// TIA Portal V19 export
DATA_BLOCK "A0301_Ribaltatore_PERS"   // DB58
// stored: MemoryReserve 100
   VAR RETAIN
      Par_Manu : "Positioning_EPOS_Machine_Par";
      Par_Aut : "A0301_Mach_Ribaltatore_Par";
   END_VAR
   VAR
      Par_Aut_Vel : Struct
         Pos1_Frw : LReal := 5000.0;
         Pos2_Frw : LReal := 5000.0;
         Pos0_Brw : LReal := 60000.0;
      END_STRUCT;
   END_VAR
   VAR RETAIN
      Pers_Data : Struct
         EncoderAbsolute_Preset_OK : Bool := TRUE;
         Persistent_ActualPosition : LReal := 2.0;
      END_STRUCT;
   END_VAR
BEGIN
   Par_Manu.PosTolerance := 0.5;
   Par_Manu.DelayInPosition := T#100MS;
   Par_Manu.Man_Vel := 15000.0;
   Par_Manu.Man_Acc := 1000.0;
   Par_Manu.Man_Dec := 1000.0;
   Par_Aut.SemiAut_Vel := 8000.0;
   Par_Aut.Aut_Vel := 8000.0;
   Par_Aut.Aut_Acc := 1000.0;
   Par_Aut.Aut_Dec := 1000.0;
   Par_Aut.Pos_0 := 2.0;
   Par_Aut.Pos_1 := 40.0;
   Par_Aut.Pos_2 := 70.0;
   Par_Aut.Pos_3 := 120.0;
END_DATA_BLOCK
